ORGANIZATION_BLOCK 主程序:OB1
TITLE=程序注释
BEGIN
Network 1 // 网络标题
// 网络注释
LD     I0.0
O      M0.0
AN     I0.1
=      M0.0
Network 2
LD     M0.0
LPS
AN     T38
TON    T37, 6000
LPP
AN     T38
TON    T38, 3000
Network 3
LD     M0.0
AN     T37
=      Q0.0
Network 4
LD     M0.0
A      T37
=      Q0.1
END_ORGANIZATION_BLOCK
SUBROUTINE_BLOCK SBR_0:SBR0
TITLE=子程序注释
BEGIN
Network 1 // 网络标题
// 网络注释
END_SUBROUTINE_BLOCK
INTERRUPT_BLOCK INT_0:INT0
TITLE=中断程序注释
BEGIN
Network 1 // 网络标题
// 网络注释
END_INTERRUPT_BLOCK
